/// This function block is a container for all linked units that are used by this unit.
/// Linked units can be addressed through their individual interface.
FUNCTION_BLOCK HandlingLinkedUnit EXTENDS HandlingContainer
VAR_INPUT

{attribute '__ZwPlcUnitEquipmentDeclaration__'} // Do not remove this attribute! It is used for code generation.
END_VAR

IF _isInitialized
THEN
  RETURN;
END_IF

{attribute '__ZwPlcUnitEquipmentImplementation__'} // Do not remove this attribute! It is used for code generation.

_isInitialized := TRUE;

END_FUNCTION_BLOCK

(* stored: Version 1.1.0.1
   POU HandlingLinkedUnit: Id {395499a4-c562-4141-9f6f-47f0f507da47}, SpecialFunc None *)
